// TIA Portal project "MP2020" (V17)

(* hardware
DEVICE "S7-1200 station_1"  S7-1200 Station
   slot 0: "Rack_0"  S7-1200 Rack  Rack  V1.0
   slot 1: "PLC_1"  CPU 1214C DC/DC/DC  6ES7 214-1AG40-0XB0  V4.5
*)

// ===== PLC "PLC_1"  CPU 1214C DC/DC/DC =====

VAR_GLOBAL   // PLC tag table "Default tag table"
   "CZ1" AT %IW64 : Int;
   "Z1" AT %Q0.0 : Bool;
   "Z2" AT %Q0.1 : Bool;
   "Z3" AT %Q0.3 : Bool;
   "M1" AT %Q0.2 : Bool;
   "Tag_1" AT %M50.0 : Bool;
   "Tag_2" AT %M50.1 : Bool;
   "Tag_3" AT %MW51 : Int;
   "Tag_4" AT %M50.2 : Bool;
   "Tag_5" AT %M50.3 : Bool;
END_VAR

DATA_BLOCK "automatyczny_mieszalnik_DB"   // DB3
{ S7_Optimized_Access := 'TRUE' }
VERSION : 0.1
// stored: InstanceOfName automatyczny_mieszalnik
"automatyczny_mieszalnik"
BEGIN
END_DATA_BLOCK

DATA_BLOCK "sterowanie_pompami_DB"   // DB5
{ S7_Optimized_Access := 'TRUE' }
VERSION : 0.1
// stored: InstanceOfName sterowanie_pompami
"sterowanie_pompami"
BEGIN
END_DATA_BLOCK

// folder: System blocks/Program resources

DATA_BLOCK "IEC_Timer_0_DB"   // DB1
{ S7_Optimized_Access := 'TRUE' }
AUTHOR : Simatic
FAMILY : IEC
NAME : IEC_TMR
VERSION : 1.0
// stored: InstanceOfName IEC_TIMER
"IEC_TIMER"
BEGIN
END_DATA_BLOCK

DATA_BLOCK "IEC_Timer_0_DB_1"   // DB2
{ S7_Optimized_Access := 'TRUE' }
AUTHOR : Simatic
FAMILY : IEC
NAME : IEC_TMR
VERSION : 1.0
// stored: InstanceOfName IEC_TIMER
"IEC_TIMER"
BEGIN
END_DATA_BLOCK

DATA_BLOCK "IEC_Timer_0_DB_2"   // DB4
{ S7_Optimized_Access := 'TRUE' }
AUTHOR : Simatic
FAMILY : IEC
NAME : IEC_TMR
VERSION : 1.0
// stored: InstanceOfName IEC_TIMER
"IEC_TIMER"
BEGIN
END_DATA_BLOCK

DATA_BLOCK "IEC_Timer_0_DB_3"   // DB6
{ S7_Optimized_Access := 'TRUE' }
AUTHOR : Simatic
FAMILY : IEC
NAME : IEC_TMR
VERSION : 1.0
// stored: InstanceOfName IEC_TIMER
"IEC_TIMER"
BEGIN
END_DATA_BLOCK

// folder: (top level)

FUNCTION_BLOCK "automatyczny_mieszalnik"   // FB1, LAD
{ S7_Optimized_Access := 'TRUE' }
VERSION : 0.1
   VAR_OUTPUT
      Z1 : Bool;
      Z2 : Bool;
      Z3 : Bool;
      step1 : Bool;
      step2 : Bool;
      step3 : Bool;
      M1 : Bool;
   END_VAR
   VAR_IN_OUT
      CZ1 : Int;
      h_cieczy : Real;
   END_VAR
   VAR
      TON_Q : Bool;
   END_VAR
   VAR_TEMP
      Sensor_norm : Real;
      norm : Real;
   END_VAR
   VAR_TEMP   // added for the SCL form of the ladder/FBD networks
      _w1 : Bool;
      _w2 : Bool;
   END_VAR
BEGIN

REGION Network 1
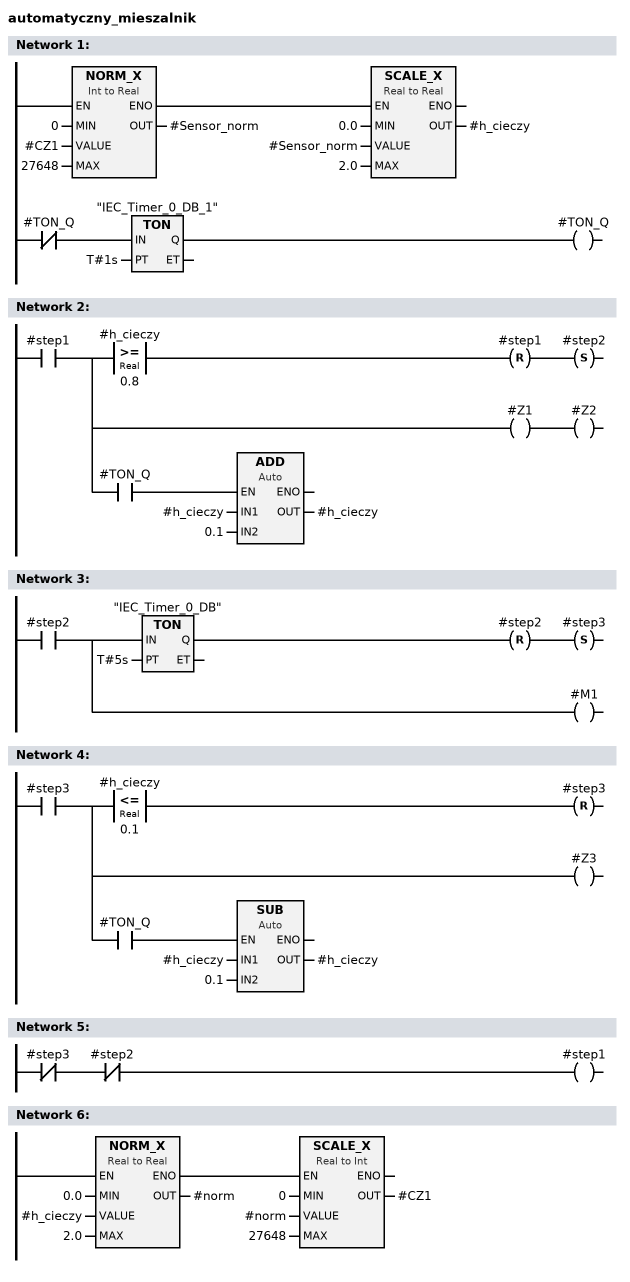
   #Sensor_norm := NORM_X(MIN := 0, VALUE := #CZ1, MAX := 27648);
   #h_cieczy := SCALE_X(MIN := 0.0, VALUE := #Sensor_norm, MAX := 2.0);
   "IEC_Timer_0_DB_1".TON(IN := NOT #TON_Q, PT := T#1s);
   #TON_Q := "IEC_Timer_0_DB_1".Q;
END_REGION

REGION Network 2
   RUNG wire#powerrail
      Contact( #step1 )
      wire#w1
      { S7_Templates := "SrcType := Real" } GE_Contact(in1 := #h_cieczy, in2 := 0.8)
      R_Coil( #step1 )
      S_Coil( #step2 )
   END_RUNG
   RUNG wire#w1
      Coil( #Z1 )
      Coil( #Z2 )
   END_RUNG
   RUNG wire#w1
      Contact( #TON_Q )
      Add(in1 := #h_cieczy, in2 := 0.1, out => #h_cieczy)
   END_RUNG
   // the same network as SCL:
   #_w1 := #step1 AND (#h_cieczy >= 0.8);
   #_w2 := #step1;
   IF #_w1 THEN
       #step1 := FALSE;
       #step2 := TRUE;
   END_IF;
   #Z1 := #_w2;
   #Z2 := #_w2;
   IF #_w2 AND #TON_Q THEN #h_cieczy := #h_cieczy + 0.1; END_IF;
END_REGION

REGION Network 3
   "IEC_Timer_0_DB".TON(IN := #step2, PT := T#5s);
   #_w1 := #step2;
   IF "IEC_Timer_0_DB".Q THEN
       #step2 := FALSE;
       #step3 := TRUE;
   END_IF;
   #M1 := #_w1;
END_REGION

REGION Network 4
   RUNG wire#powerrail
      Contact( #step3 )
      wire#w1
      { S7_Templates := "SrcType := Real" } LE_Contact(in1 := #h_cieczy, in2 := 0.1)
      R_Coil( #step3 )
   END_RUNG
   RUNG wire#w1
      Coil( #Z3 )
   END_RUNG
   RUNG wire#w1
      Contact( #TON_Q )
      Sub(in1 := #h_cieczy, in2 := 0.1, out => #h_cieczy)
   END_RUNG
   // the same network as SCL:
   #_w1 := #step3;
   IF #step3 AND (#h_cieczy <= 0.1) THEN #step3 := FALSE; END_IF;
   #Z3 := #_w1;
   IF #_w1 AND #TON_Q THEN #h_cieczy := #h_cieczy - 0.1; END_IF;
END_REGION

REGION Network 5
   RUNG wire#powerrail
      I_Contact( #step3 )
      I_Contact( #step2 )
      Coil( #step1 )
   END_RUNG
   // the same network as SCL:
   #step1 := NOT #step3 AND NOT #step2;
END_REGION

REGION Network 6
   RUNG wire#powerrail
      { S7_Templates := "[SrcType := Real, DestType := Real]" } Normalize(min := 0.0, value := #h_cieczy, max := 2.0, out => #norm)
      { S7_Templates := "[SrcType := Real, DestType := Int]" } Scale(min := 0, value := #norm, max := 27648, out => #CZ1)
   END_RUNG
   // the same network as SCL:
   #norm := NORM_X(MIN := 0.0, VALUE := #h_cieczy, MAX := 2.0);
   #CZ1 := SCALE_X(MIN := 0, VALUE := #norm, MAX := 27648);
END_REGION
END_FUNCTION_BLOCK

FUNCTION_BLOCK "sterowanie_pompami"   // FB2, LAD
{ S7_Optimized_Access := 'TRUE' }
VERSION : 0.1
   VAR_INPUT
      failurePump1 : Bool;
      failurePump2 : Bool;
      valveOpenConf11 : Bool;
      valveCloseConf11 : Bool;
      valveOpenConf12 : Bool;
      valveCloseConf12 : Bool;
      valveOpenConf21 : Bool;
      valveCloseConf21 : Bool;
      valveOpenConf22 : Bool;
      valveCloseConf22 : Bool;
      pressureValue : Int;
   END_VAR
   VAR_OUTPUT
      pump1 : Bool;
      pump2 : Bool;
      valveOpen1 : Bool;
      valveClose1 : Bool;
      valveOpen2 : Bool;
      valveClose2 : Bool;
   END_VAR
   VAR
      M0 : Bool;
      M1 : Bool;
      M2 : Bool;
   END_VAR
   VAR_TEMP
      pressure_bar : Real;
   END_VAR
   VAR_TEMP   // added for the SCL form of the ladder/FBD networks
      _w1 : Bool;
   END_VAR
BEGIN

REGION Network 1
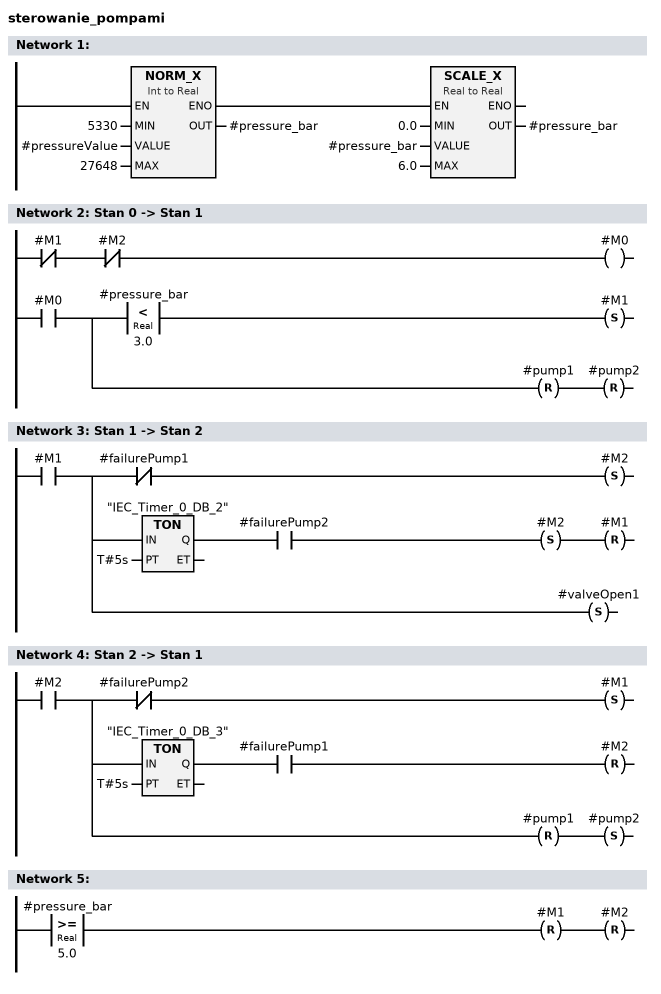
   RUNG wire#powerrail
      { S7_Templates := "[SrcType := Int, DestType := Real]" } Normalize(min := 5330, value := #pressureValue, max := 27648, out => #pressure_bar)
      { S7_Templates := "[SrcType := Real, DestType := Real]" } Scale(min := 0.0, value := #pressure_bar, max := 6.0, out => #pressure_bar)
   END_RUNG
   // the same network as SCL:
   #pressure_bar := NORM_X(MIN := 5330, VALUE := #pressureValue, MAX := 27648);
   #pressure_bar := SCALE_X(MIN := 0.0, VALUE := #pressure_bar, MAX := 6.0);
END_REGION

REGION Network 2: Stan 0 -> Stan 1
   RUNG wire#powerrail
      I_Contact( #M1 )
      I_Contact( #M2 )
      Coil( #M0 )
   END_RUNG
   RUNG wire#powerrail
      Contact( #M0 )
      wire#w1
      { S7_Templates := "SrcType := Real" } LT_Contact(in1 := #pressure_bar, in2 := 3.0)
      S_Coil( #M1 )
   END_RUNG
   RUNG wire#w1
      R_Coil( #pump1 )
      R_Coil( #pump2 )
   END_RUNG
   // the same network as SCL:
   #M0 := NOT #M1 AND NOT #M2;
   IF #M0 AND (#pressure_bar < 3.0) THEN #M1 := TRUE; END_IF;
   IF #M0 THEN
       #pump1 := FALSE;
       #pump2 := FALSE;
   END_IF;
END_REGION

REGION Network 3: Stan 1 -> Stan 2
   IF #M1 AND NOT #failurePump1 THEN #M2 := TRUE; END_IF;
   "IEC_Timer_0_DB_2".TON(IN := #M1, PT := T#5s);
   IF "IEC_Timer_0_DB_2".Q AND #failurePump2 THEN #M2 := TRUE; END_IF;
   #_w1 := #M1;
   IF "IEC_Timer_0_DB_2".Q AND #failurePump2 THEN #M1 := FALSE; END_IF;
   IF #_w1 THEN #valveOpen1 := TRUE; END_IF;
END_REGION

REGION Network 4: Stan 2 -> Stan 1
   IF #M2 AND NOT #failurePump2 THEN #M1 := TRUE; END_IF;
   "IEC_Timer_0_DB_3".TON(IN := #M2, PT := T#5s);
   #_w1 := #M2;
   IF "IEC_Timer_0_DB_3".Q AND #failurePump1 THEN #M2 := FALSE; END_IF;
   IF #_w1 THEN
       #pump1 := FALSE;
       #pump2 := TRUE;
   END_IF;
END_REGION

REGION Network 5
   RUNG wire#powerrail
      { S7_Templates := "SrcType := Real" } GE_Contact(in1 := #pressure_bar, in2 := 5.0)
      R_Coil( #M1 )
      R_Coil( #M2 )
   END_RUNG
   // the same network as SCL:
   IF #pressure_bar >= 5.0 THEN
       #M1 := FALSE;
       #M2 := FALSE;
   END_IF;
END_REGION
END_FUNCTION_BLOCK

ORGANIZATION_BLOCK "Main"   // OB1, LAD, ProgramCycle
TITLE = "Main Program Sweep (Cycle)"
{ S7_Optimized_Access := 'TRUE' }
VERSION : 0.1
   VAR_INPUT
      Initial_Call : Bool;   // Initial call of this OB
      Remanence : Bool;   // =True, if remanent data are available
   END_VAR
BEGIN

REGION Network 1
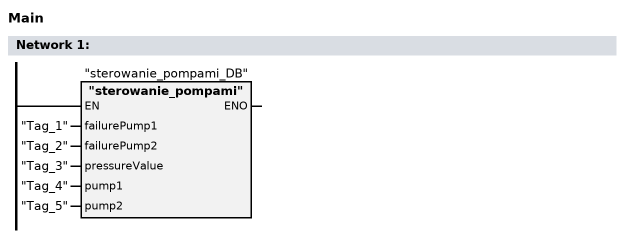
   RUNG wire#powerrail
      "sterowanie_pompami_DB"(failurePump1 := "Tag_1", failurePump2 := "Tag_2", pressureValue := "Tag_3", pump1 := "Tag_4", pump2 := "Tag_5")
   END_RUNG
   // the same network as SCL:
   "sterowanie_pompami_DB"(failurePump1 := "Tag_1",   // "sterowanie_pompami"
                           failurePump2 := "Tag_2",
                           pressureValue := "Tag_3",
                           pump1 := "Tag_4",
                           pump2 := "Tag_5");
END_REGION
END_ORGANIZATION_BLOCK